{attribute 'qualified_only'}
{attribute 'strict'}
{attribute 'to_string'}
TYPE E_AlarmSeverity :
(
    Information := 0,
    Warning := 10,
    Fault := 20,
    SafetyStop := 30
);
END_TYPE

(* stored: Version 1.1.0.1, ProductVersion 3.1.4026.18
   DUT E_AlarmSeverity: Id {fbfb399f-be25-4f59-a990-3f98c0d98479} *)
